FUNCTION F_GetSymbolName : string(255)
VAR_INPUT
	Symobl:				ANY;
END_VAR
VAR
	fbJsonReadWriteDataType: FB_JsonReadWriteDataType;
END_VAR

F_GetSymbolName:= fbJsonReadWriteDataType.GetDatatypeNameByAddress(Symobl.diSize, Symobl.pValue);

END_FUNCTION

(* stored: Version 1.1.0.1
   POU F_GetSymbolName: Id {32af0d2c-87c0-45e5-8b3b-e3d3a368786a}, SpecialFunc None *)
